FUNCTION TransferMotorDataToProxy : BOOL
VAR_INPUT
	mp: POINTER TO MotorProxy;
	
END_VAR
VAR
	
	prox: MotorProxy;
	moto: Motor;



END_VAR


	
	prox := mp^;
	mp := prox.motorPtr^;
	
	prox.encoder := moto.encoder;
	prox.IsAxisSelected := moto.isAxisSelected;
	prox.status := moto.status;

END_FUNCTION

(* stored: Version 1.1.0.1, ProductVersion 3.1.4024.13
   POU TransferMotorDataToProxy: Id {a81a26a7-a9c2-4643-a97f-52109abaf75f}, SpecialFunc None *)
